{attribute 'qualified_only'}
VAR_GLOBAL
	valve01: DUT_VALVE;
	io_values: DUT_IO_Valve;
END_VAR

(* stored: Version 1.1.0.1, ProductVersion 3.1.4024.12
   GVL GVL_VCM: Id {fa8f2333-72af-4d12-8190-dfd5666fec84} *)
